(* PLC project single_acting_jack, Dassault Systèmes ControlBuild 2024x *)
(* stored: creationDateTime 2023-10-03T11:13:08-01:00 *)

(* This module simulates a single-acting jack driven by a three-way, two positions control valve *)
FUNCTION_BLOCK equipment_library.single_acting_jack
  VAR_INPUT
    energy : BOOL := true;
    cmdSupply : BOOL := true;
    sensorSupply : BOOL := true;
  END_VAR
  VAR_INPUT
    valveWork : BOOL := false;
  END_VAR
  VAR_OUTPUT
    outletSensor : BOOL := false;
    inletSensor : BOOL := false;
  END_VAR
  VAR_OUTPUT
    rodPosition : REAL := 0.0;
    rodPercent : REAL := 0.0;
    incrementValue : REAL := 0.0;
  END_VAR
  VAR
    slidePosition : DINT := 0;
    pipeWork : BOOL := false;
    pipeRest : BOOL := false;
    increment : REAL := 0.0;
  END_VAR
  VAR CONSTANT
    outletSensorLogic : BOOL := true;
    inletSensorLogic : BOOL := true;
    rodLength : REAL := 1000.0;
    time2extend : REAL := 2.0;
  END_VAR
  VAR
    d_locking : BOOL := false;
    v_d_locking : REAL := 2.0;
    d_inletSensor : BOOL := false;
    v_d_inletSensor : BOOL := false;
    d_outletSensor : BOOL := false;
    v_d_outletSensor : BOOL := false;
  END_VAR


ACTION C_source_code:
/* ----------------------------------------------------------------	*/
/* Type : Model of Operative Behaviour					*/
/* Category :  Associations - Jacks					*/
/* Author : Dassault Systemes						*/
/* Update date : June 2018							*/
/* ----------------------------------------------------------------	*/
/* This module simulates a single-acting jack driven by a   		*/
/* three-way, two positions control valve .				*/
/* ----------------------------------------------------------------	*/

/* ----------------------------------------------------------------	*/
/* Management of orders from Control Part					*/
/*	if there is no power supply for command the solenoid 		*/
/*     control valve doesn't understand the control order.		*/
/* ----------------------------------------------------------------	*/
if (cmdSupply && valveWork) slidePosition = 1;
else slidePosition = 0;

/* ----------------------------------------------------------------	*/
/* Calculation of the on-state of the energy in the pipes		*/
/*     if there is no energy in input, pipes are not 			*/
/*	   under pressure.							*/
/* ----------------------------------------------------------------	*/
pipeWork = (slidePosition==1) & energy;
pipeRest = 0;

/* ----------------------------------------------------------------	*/
/* Management of the rod evolution						*/
/* ----------------------------------------------------------------	*/
incrementValue = 0;
if (! d_locking)  {
	if (time2extend > 0.0)
		increment = (rodLength/time2extend)*(CLOCK_PERIOD/1000000);
	if (pipeWork && ! pipeRest) {
		if ( rodPosition < rodLength ) {
			(rodPosition) += increment;
			incrementValue = increment;
		}
		if ( rodPosition > rodLength ) {
			incrementValue -= rodPosition - rodLength;
			rodPosition = rodLength;
		}
	}
	else {
		if ( rodPosition > 0 ) {
			(rodPosition) -= increment;
			incrementValue = increment * -1.0;
		}
		if ( rodPosition < 0.0 ) {
			incrementValue -= rodPosition;
			rodPosition = 0.0;
		}
	}
}

/* ----------------------------------------------------------------	*/
/* Calculation of the rod position in percentage			*/
/* ----------------------------------------------------------------	*/
rodPercent = ((rodPosition/rodLength)*100);

/* ----------------------------------------------------------------	*/
/* Management of the sensors state						*/
/* ----------------------------------------------------------------	*/
if (d_outletSensor) outletSensor = v_d_outletSensor;
else
	outletSensor = ((rodPosition >= rodLength) ^ ! outletSensorLogic) && sensorSupply;


if (d_inletSensor) inletSensor = v_d_inletSensor;
else
	inletSensor = ((rodPosition <= 0) ^ ! inletSensorLogic) && sensorSupply;
END_ACTION
END_FUNCTION_BLOCK
